(* IEC 61131-3 sources: CodesysTest/alpha/export/FBs/Unused/MotorizedSealFlattenersFB.pou/Ready.prop, 1 file *)

(* ---- Set.pm.st ---- *)
(*#-#-#-#-#-#-#-#-#-#---Declaration---#-#-#-#-#-#-#-#-#-#-#-#-#*)

VAR
END_VAR
(*#-#-#-#-#-#-#-#-#-#---Implementation---#-#-#-#-#-#-#-#-#-#-#-#-#*)

_ready := Ready;
